ABB RobotStudio station: Oke_Iyanuoluwa.rspag

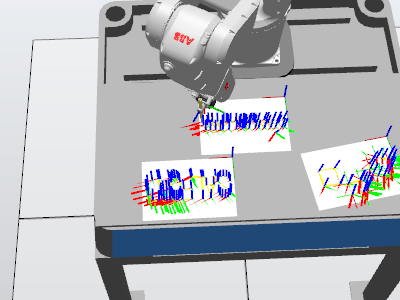
--- station ---
Station Project8 (saved by RobotStudio 24.1.10713.1)
Controller IRB1200_5_90, task T_ROB1: task frame (RAPID world) sits at (0, 233, 928) mm, rotated rx 0 ry 0 rz -90 deg in the station
Controller IRB1200_5_90
  mechanical unit ROB_1: IRB1200FPL_5_90_STD_02, 6 joints, base frame (0, 0, 0) mm
Layout (positions relative to the parent item):
  - IRB1200FPL_5_90_STD_02 [mechanism, from %ABB.RobotStudio.Models.IRB1200%\IRB1200FPL_5_90_STD_02.rslib] at (0, 233, 928) mm, rotated rx 0 ry 0 rz -90 deg; joint values [-0.5118, 1.2481, 0.7456, 0.0144, -1.9002, 0.0022] (rad or m)
  - Hardware [part], size 1120 x 955 x 931 mm
  - Pen for irb1200_2 [part] at (-177.12, -80.05, 1033) mm, rotated rx -87.72 ry 84.63 rz 62.19 deg, size 168 x 34 x 40 mm
  - IYANU2 [part] at (97, -87.87, 931) mm, rotated rx 0 ry 0 rz 180 deg, size 276.3 x 33.8 x 1 mm
Attachment: Pen for irb1200_2 is attached to IRB1200FPL_5_90_STD_02 / Link6
Targets, tools, work objects and paths stored in the station and not in the controller backup, written as RAPID:
! task T_ROB1
MODULE Module1
  PROC Shape_CircleCopy()
    MoveJ il_186,v100,fine,toolPen\WObj:=wobjShapes;
    MoveL il_187,v100,fine,toolPen\WObj:=wobjShapes;
    MoveL il_188,v100,fine,toolPen\WObj:=wobjShapes;
    MoveL il_189,v100,fine,toolPen\WObj:=wobjShapes;
    MoveL il_190,v100,fine,toolPen\WObj:=wobjShapes;
    MoveL il_191,v100,fine,toolPen\WObj:=wobjShapes;
    MoveL il_192,v100,fine,toolPen\WObj:=wobjShapes;
    MoveL il_193,v100,fine,toolPen\WObj:=wobjShapes;
    MoveL il_194,v100,fine,toolPen\WObj:=wobjShapes;
    MoveL il_195,v100,fine,toolPen\WObj:=wobjShapes;
    MoveL il_196,v100,fine,toolPen\WObj:=wobjShapes;
    MoveL il_197,v100,fine,toolPen\WObj:=wobjShapes;
    MoveL il_198,v100,fine,toolPen\WObj:=wobjShapes;
    MoveL il_199,v100,fine,toolPen\WObj:=wobjShapes;
  ENDPROC
ENDMODULE


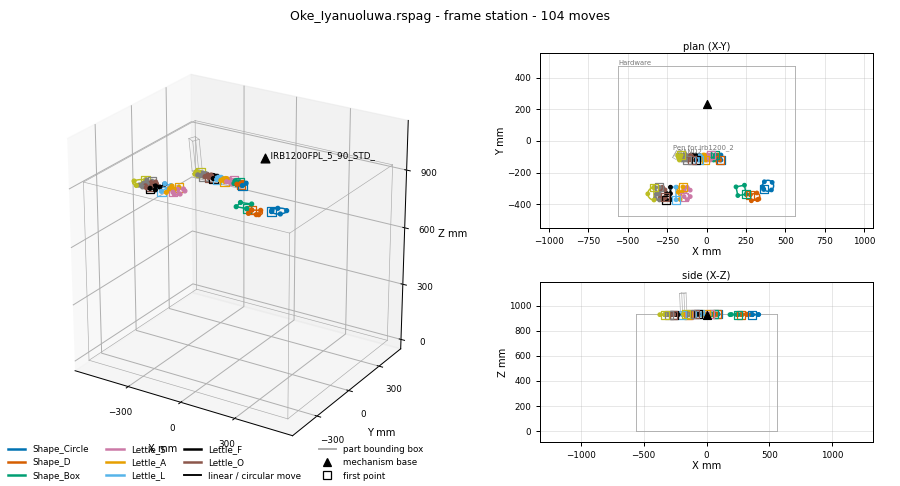
[picture p0: tool path of Oke_Iyanuoluwa.rspag in frame station, 104 of 104 moves have a stored position in this frame; points joined in program order, loops and branches not executed]
--- Controller Data/IRB1200_5_90/RAPID/TASK1/PROGMOD/Module1.mod ---
MODULE Module1
	TASK PERS tooldata toolPen:=[TRUE,[[100,0,20],[0.653281482,0.27059805,-0.653281482,-0.27059805]],[0.1,[50,0,10],[1,0,0,0],0,0,0]];
	TASK PERS wobjdata wobjShapes:=[FALSE,TRUE,"",[[403.87242208,428.126413661,0.1],[0.765935658,-0.001715767,0.001440186,-0.64291333]],[[0,0,0],[1,0,0,0]]];
	TASK PERS wobjdata wobjSalford:=[FALSE,TRUE,"",[[459.660289856,-90.375541036,0.1],[0.711712441,0,0,-0.702470925]],[[0,0,0],[1,0,0,0]]];
	TASK PERS wobjdata wobjName:=[FALSE,TRUE,"",[[234.420012927,103.808224608,3],[0.710975028,0,0,-0.703217256]],[[0,0,0],[1,0,0,0]]];
	VAR num MyChoice:=0;
    CONST robtarget Target_10:=[[511.467625969,422.116161374,0.1],[0,-0.087155742,0.996194698,0],[0,0,0,0],[9E+09,9E+09,9E+09,9E+09,9E+09,9E+09]];
    CONST robtarget Target_20:=[[485.422114903,400.261382644,0.1],[0,-0.573576436,0.819152044,0],[0,0,0,0],[9E+09,9E+09,9E+09,9E+09,9E+09,9E+09]];
    CONST robtarget Target_30:=[[491.326152944,366.777919042,0.1],[0,0.906307787,-0.422618262,0],[0,0,0,0],[9E+09,9E+09,9E+09,9E+09,9E+09,9E+09]];
    CONST robtarget Target_40:=[[523.275702051,355.149234169,0.1],[0,0.996194698,0.087155742,0],[0,0,0,0],[9E+09,9E+09,9E+09,9E+09,9E+09,9E+09]];
    CONST robtarget Target_50:=[[549.321213117,377.004012898,0.1],[0,0.819152044,0.573576436,0],[0,0,0,0],[9E+09,9E+09,9E+09,9E+09,9E+09,9E+09]];
    CONST robtarget Target_60:=[[543.417175076,410.4874765,0.1],[0,0.422618262,0.906307787,0],[0,0,0,0],[9E+09,9E+09,9E+09,9E+09,9E+09,9E+09]];
    CONST robtarget Target_70:=[[511.467625969,422.116161374,0.1],[0,-0.087155742,0.996194698,0],[0,0,0,0],[9E+09,9E+09,9E+09,9E+09,9E+09,9E+09]];
    CONST robtarget Target_80:=[[511.467625969,422.116161374,0.1],[0,-0.087155742,0.996194698,0],[0,0,0,0],[9E+09,9E+09,9E+09,9E+09,9E+09,9E+09]];
    CONST robtarget Target_90:=[[483.888200408,382.72865973,0.1],[0,0.766044443,-0.642787609,0],[0,0,0,0],[9E+09,9E+09,9E+09,9E+09,9E+09,9E+09]];
    CONST robtarget Target_100:=[[523.275702051,355.149234169,0.1],[0,0.996194698,0.087155742,0],[0,0,0,0],[9E+09,9E+09,9E+09,9E+09,9E+09,9E+09]];
    CONST robtarget Target_110:=[[550.855127612,394.536735812,0.1],[0,0.642787609,0.766044443,0],[0,0,0,0],[9E+09,9E+09,9E+09,9E+09,9E+09,9E+09]];
    CONST robtarget Target_120:=[[511.467625969,422.116161374,0.1],[0,-0.087155742,0.996194698,0],[0,0,0,0],[9E+09,9E+09,9E+09,9E+09,9E+09,9E+09]];
    CONST robtarget Target_130:=[[24.567771359,104.924042365,0.470081631],[0.001584245,-0.707222542,0.706987453,0.001583718],[0,0,0,0],[9E+09,9E+09,9E+09,9E+09,9E+09,9E+09]];
    CONST robtarget Target_140:=[[92.567767601,104.946649893,0.470182963],[0.001584245,-0.707222542,0.706987453,0.001583718],[0,0,0,0],[9E+09,9E+09,9E+09,9E+09,9E+09,9E+09]];
    CONST robtarget Target_150:=[[31.05454894,124.910653298,0.569625926],[0.001995763,-0.890928808,-0.454137469,-0.001017311],[0,0,0,0],[9E+09,9E+09,9E+09,9E+09,9E+09,9E+09]];
    CONST robtarget Target_160:=[[69.063596083,137.274389626,0.625018071],[0.002212567,-0.987711853,0.156269884,0.000350059],[0,0,0,0],[9E+09,9E+09,9E+09,9E+09,9E+09,9E+09]];
    CONST robtarget Target_170:=[[92.567767601,104.946605091,0.480182863],[0.001584245,-0.707222542,0.706987453,0.001583718],[0,0,0,0],[9E+09,9E+09,9E+09,9E+09,9E+09,9E+09]];
    CONST robtarget Target_180:=[[138.556128715,139.961590026,0.627057236],[0.002240087,-0.999997477,-0.000166233,-0.000000373],[0,0,0,0],[9E+09,9E+09,9E+09,9E+09,9E+09,9E+09]];
    CONST robtarget Target_190:=[[178.556126504,139.974888571,0.627116843],[0.002240087,-0.999997477,-0.000166233,-0.000000373],[0,0,0,0],[9E+09,9E+09,9E+09,9E+09,9E+09,9E+09]];
    CONST robtarget Target_200:=[[178.542827825,179.974484922,0.806323386],[0.001583718,-0.706987453,-0.707222542,-0.001584245],[0,0,0,0],[9E+09,9E+09,9E+09,9E+09,9E+09,9E+09]];
    CONST robtarget Target_210:=[[138.542830036,179.961186376,0.806263778],[0.000000373,-0.000166233,0.999997477,0.002240087],[0,0,0,0],[9E+09,9E+09,9E+09,9E+09,9E+09,9E+09]];
    CONST robtarget Target_220:=[[118.549480481,159.954738929,0.716630704],[0.001584245,-0.707222542,0.706987453,0.001583718],[0,0,0,0],[9E+09,9E+09,9E+09,9E+09,9E+09,9E+09]];
    CONST robtarget Target_230:=[[124.412046326,145.814693543,0.653280352],[0.002069714,-0.923940816,0.382528888,0.0008569],[0,0,0,0],[9E+09,9E+09,9E+09,9E+09,9E+09,9E+09]];
    CONST robtarget Target_240:=[[138.556128715,139.961590026,0.627057236],[0.002240087,-0.999997477,-0.000166233,-0.000000373],[0,0,0,0],[9E+09,9E+09,9E+09,9E+09,9E+09,9E+09]];
	CONST zonedata zone1:=[FALSE,50,75,75,7.5,75,7.5];
    !***********************************************************
    !
    ! Module:  Module1
    !
    ! Description:
    !   <Insert description here>
    !
    ! Author: sdp562
    !
    ! Version: 1.0
    !
    !***********************************************************


    !***********************************************************
    !
    ! Procedure main
    !
    !   This is the entry point of your program
    !
    !***********************************************************
    PROC main()
        TPErase;
        TPWrite "ABB RobotStudio Assignment - Oke Iyanuoluwa E.";
        TPReadFK MyChoice, "What will you like to draw/write?", "Shapes", "Salford", "MyName", "All of the above", stEmpty;
        TEST MyChoice
        CASE 1:
        	Shapes;
        CASE 2:
        	Salford;
        CASE 3:
        	MyName;
        CASE 4:
        	All;
        ENDTEST
    ENDPROC
	PROC Shapes()
		Shape_Circle;
		WaitTime 2;
		Shape_D;
		WaitTime 2;
		Shape_Box;
	ENDPROC
	PROC Salford()
		Lettle_S;
		Lettle_A;
		Lettle_L;
		Lettle_F;
		Lettle_O;
		Lettle_R;
		Lettle_D;
	ENDPROC
	PROC MyName()
		Letter_I;
		Letter_Y;
		Letter_A2;
		Letter_N;
		Letter_U;
		Letter_O2;
		Letter_L2;
		Letter_U2;
		Lettter_W;
		Letter_A3;
	ENDPROC
	PROC All()
		Shapes;
		WaitTime 2;
		Salford;
		WaitTime 2;
		MyName;
	ENDPROC
	PROC Shape_Circle()
		MoveJ [[88.31,121.43,0.9],[0.824392,-0.00205287,-0.000613241,0.566015],[0,-1,-1,1],[9E+09,9E+09,9E+09,9E+09,9E+09,9E+09]], v100, fine, toolPen\WObj:=wobjShapes;
		MoveC [[92.64,104.84,0.86],[0.823057,-0.0156436,0.0018724,0.567741],[0,-1,-1,1],[9E+09,9E+09,9E+09,9E+09,9E+09,9E+09]], [[75.99,75.44,-0.17],[0.809935,-0.0315414,0.00398667,0.585658],[0,-1,-1,1],[9E+09,9E+09,9E+09,9E+09,9E+09,9E+09]], v100, z10, toolPen\WObj:=wobjShapes;
		MoveC [[58.82,69.88,0.86],[0.801435,-0.0289154,0.00307954,0.597375],[0,-1,-1,1],[9E+09,9E+09,9E+09,9E+09,9E+09,9E+09]], [[27.99,88.04,1.08],[0.793128,-0.0040181,-0.000672612,0.609041],[0,-1,-1,1],[9E+09,9E+09,9E+09,9E+09,9E+09,9E+09]], v100, z10, toolPen\WObj:=wobjShapes;
		MoveC [[22.52,102.18,2.75],[0.794173,0.00861844,-0.00234434,0.607627],[0,-1,-1,1],[9E+09,9E+09,9E+09,9E+09,9E+09,9E+09]], [[41.05,134.37,1.12],[0.808041,0.0241329,-0.00490428,0.588611],[0,-1,-1,1],[9E+09,9E+09,9E+09,9E+09,9E+09,9E+09]], v100, z10, toolPen\WObj:=wobjShapes;
		MoveC [[57.78,139.03,0.62],[0.815418,0.0212852,-0.00468144,0.578462],[0,-1,-1,1],[9E+09,9E+09,9E+09,9E+09,9E+09,9E+09]], [[88.04,122.04,0.46],[0.826354,-0.00524432,0.00563442,0.563098],[0,0,0,1],[9E+09,9E+09,9E+09,9E+09,9E+09,9E+09]], v100, z10, toolPen\WObj:=wobjShapes;
		MoveL [[92.89,104.88,1.07],[0.825128,-0.0192408,0.00814959,0.564559],[0,0,0,1],[9E+09,9E+09,9E+09,9E+09,9E+09,9E+09]], v100, fine, toolPen\WObj:=wobjShapes;
	ENDPROC
	PROC Shape_D()
		MoveJ [[178.33,139.97,0.82],[0.862322,-0.0124094,0.00252986,0.506202],[0,-1,-1,1],[9E+09,9E+09,9E+09,9E+09,9E+09,9E+09]], v100, fine, toolPen\WObj:=wobjShapes;
		MoveL [[135.18,137.21,5.02],[0.84537,-0.00306398,-0.00014847,0.534173],[0,-1,-1,1],[9E+09,9E+09,9E+09,9E+09,9E+09,9E+09]], v100, fine, toolPen\WObj:=wobjShapes;
		MoveC [[122.15,149.76,0.21],[0.842062,0.00867023,-0.00276849,0.539304],[0,-1,-1,1],[9E+09,9E+09,9E+09,9E+09,9E+09,9E+09]],[[129.21,176.92,0.5],[0.84799,0.027547,-0.00720098,0.529246],[0,-1,-1,1],[9E+09,9E+09,9E+09,9E+09,9E+09,9E+09]],v100,z10,toolPen\WObj:=wobjShapes;
		MoveL [[139.7,179.86,0.26],[0.852174,0.027013,-0.00727031,0.52251],[0,-1,-1,1],[9E+09,9E+09,9E+09,9E+09,9E+09,9E+09]],v100,fine,toolPen\WObj:=wobjShapes;
		MoveL [[177.84,179.74,0.48],[0.866093,0.0181024,-0.00553464,0.499525],[0,-1,-1,1],[9E+09,9E+09,9E+09,9E+09,9E+09,9E+09]], v100, fine, toolPen\WObj:=wobjShapes;
		MoveL [[177.74,140.56,0.46],[0.862166,-0.0119302,0.00239961,0.50648],[0,-1,-1,1],[9E+09,9E+09,9E+09,9E+09,9E+09,9E+09]], v100, fine, toolPen\WObj:=wobjShapes;
	ENDPROC
	PROC Shape_Box()
		MoveJ [[203.77,133.76,1.09],[0.871331,-0.0217624,0.00553483,0.490182],[0,-1,-1,1],[9E+09,9E+09,9E+09,9E+09,9E+09,9E+09]], v100, fine, toolPen\WObj:=wobjShapes;
		MoveL [[256.61,132.45,1.81],[0.890805,-0.0302163,0.00946486,0.45328],[0,-1,-1,1],[9E+09,9E+09,9E+09,9E+09,9E+09,9E+09]], v100, fine, toolPen\WObj:=wobjShapes;
		MoveL [[258.42,76.19,0.13],[0.885765,-0.0735338,0.0230334,0.457692],[0,-1,-1,1],[9E+09,9E+09,9E+09,9E+09,9E+09,9E+09]], v100, fine, toolPen\WObj:=wobjShapes;
		MoveL [[203.82,75.03,0.64],[0.863466,-0.0662649,0.0170718,0.499743],[0,-1,-1,1],[9E+09,9E+09,9E+09,9E+09,9E+09,9E+09]], v100, fine, toolPen\WObj:=wobjShapes;
		MoveL [[203.76,134.33,0.29],[0.871385,-0.0215486,0.00547808,0.490096],[0,-1,-1,1],[9E+09,9E+09,9E+09,9E+09,9E+09,9E+09]], v100, fine, toolPen\WObj:=wobjShapes;
	ENDPROC
	PROC Lettle_S()
		MoveJ [[53.37,125.02,0.18],[0.963615,-0.0368758,0.0208919,0.263911],[-1,-1,-1,1],[9E+09,9E+09,9E+09,9E+09,9E+09,9E+09]], v100, fine, toolPen\WObj:=wobjSalford;
		MoveC [[49.77,135.43,-0.38],[0.962565,-0.0306315,0.0171276,0.268771],[-1,-1,-1,1],[9E+09,9E+09,9E+09,9E+09,9E+09,9E+09]],[[33.43,144.4,0.22],[0.958673,-0.0271208,0.0146305,0.282836],[-1,-1,-1,1],[9E+09,9E+09,9E+09,9E+09,9E+09,9E+09]],v100,z10,toolPen\WObj:=wobjSalford;
		MoveC [[24.37,142.14,-0.7],[0.956604,-0.0303515,0.0161234,0.289358],[-1,-1,-1,1],[9E+09,9E+09,9E+09,9E+09,9E+09,9E+09]],[[14.25,125.41,-0.8],[0.954383,-0.0435766,0.0229035,0.294497],[-1,-1,-1,1],[9E+09,9E+09,9E+09,9E+09,9E+09,9E+09]],v100,z10,toolPen\WObj:=wobjSalford;
		MoveL [[52.61,85.48,0.05],[0.963977,-0.0634662,0.0367473,0.255677],[-1,-1,-1,1],[9E+09,9E+09,9E+09,9E+09,9E+09,9E+09]], v100, fine, toolPen\WObj:=wobjSalford;
		MoveC [[50.58,75.89,-0.86],[0.963497,-0.070496,0.0408837,0.255014],[-1,-1,-1,1],[9E+09,9E+09,9E+09,9E+09,9E+09,9E+09]], [[33.64,65.84,-0.65],[0.959249,-0.0807602,0.0455016,0.266923],[-1,-1,-1,1],[9E+09,9E+09,9E+09,9E+09,9E+09,9E+09]], v100, z10, toolPen\WObj:=wobjSalford;
		MoveC [[24.01,68.64,-0.57],[0.956773,-0.0808116,0.0445486,0.275809],[-1,-1,-1,1],[9E+09,9E+09,9E+09,9E+09,9E+09,9E+09]], [[13.83,84.72,0.25],[0.954272,-0.0714944,0.0382654,0.28773],[-1,-1,-1,1],[9E+09,9E+09,9E+09,9E+09,9E+09,9E+09]], v100, z10, toolPen\WObj:=wobjSalford;
	ENDPROC
	PROC Lettle_A()
		MoveJ [[59.29,63.59,0.56],[0.965584,-0.0761666,0.0452825,0.244532],[-1,-1,-1,1],[9E+09,9E+09,9E+09,9E+09,9E+09,9E+09]], v100, fine, toolPen\WObj:=wobjSalford;
		MoveL [[78.48,142.56,0.21],[0.968312,-0.0201088,0.0117518,0.248656],[-1,-1,-1,1],[9E+09,9E+09,9E+09,9E+09,9E+09,9E+09]], v100, fine, toolPen\WObj:=wobjSalford;
		MoveL [[97.6,65.33,0.08],[0.973898,-0.0654568,0.0418275,0.213279],[-1,-1,-1,1],[9E+09,9E+09,9E+09,9E+09,9E+09,9E+09]], v100, fine, toolPen\WObj:=wobjSalford;
		MoveL [[89.96,96.6,-0.46],[0.971904,-0.0478143,0.0294838,0.228577],[-1,-1,-1,1],[9E+09,9E+09,9E+09,9E+09,9E+09,9E+09]], v100, fine, toolPen\WObj:=wobjSalford;
		MoveL [[66.19,95.41,0.1],[0.966964,-0.0539454,0.0318698,0.247092],[-1,-1,-1,1],[9E+09,9E+09,9E+09,9E+09,9E+09,9E+09]], v100, fine, toolPen\WObj:=wobjSalford;
	ENDPROC
	PROC Lettle_L()
		MoveJ [[104.07,144.38,0.11],[0.97299,-0.0134348,0.00814553,0.230311],[-1,-1,-1,1],[9E+09,9E+09,9E+09,9E+09,9E+09,9E+09]], v100, fine, toolPen\WObj:=wobjSalford;
		MoveL [[104.04,64.44,0.45],[0.975186,-0.0641498,0.0415036,0.207783],[-1,-1,-1,1],[9E+09,9E+09,9E+09,9E+09,9E+09,9E+09]], v100, fine, toolPen\WObj:=wobjSalford;
		MoveL [[137.15,65.07,3.55],[0.98121,-0.0534444,0.03662,0.181739],[-1,-1,-1,1],[9E+09,9E+09,9E+09,9E+09,9E+09,9E+09]], v100, fine, toolPen\WObj:=wobjSalford;
	ENDPROC
	PROC Lettle_F()
		MoveJ [[168.45,142.39,0.47],[0.982868,0.00146233,-0.00116288,0.184302],[-1,-1,-1,1],[9E+09,9E+09,9E+09,9E+09,9E+09,9E+09]], v100, fine, toolPen\WObj:=wobjSalford;
		MoveL [[138.89,143.45,-0.22],[0.978706,-0.00579302,0.00363048,0.205151],[-1,-1,-1,1],[9E+09,9E+09,9E+09,9E+09,9E+09,9E+09]], v100, fine, toolPen\WObj:=wobjSalford;
		MoveL [[138.71,64.53,0.13],[0.981408,-0.0541674,0.0372314,0.180327],[-1,-1,-1,1],[9E+09,9E+09,9E+09,9E+09,9E+09,9E+09]], v100, fine, toolPen\WObj:=wobjSalford;
		MoveL [[139.2,104.9,0.04],[0.980441,-0.0297577,0.0198081,0.19354],[-1,-1,-1,1],[9E+09,9E+09,9E+09,9E+09,9E+09,9E+09]], v100, fine, toolPen\WObj:=wobjSalford;
		MoveL [[163.35,104.29,0.13],[0.98403,-0.0232892,0.0160867,0.175739],[-1,-1,-1,1],[9E+09,9E+09,9E+09,9E+09,9E+09,9E+09]], v100, fine, toolPen\WObj:=wobjSalford;
	ENDPROC
	PROC Lettle_O()
		MoveJ [[173.96,128.87,0.16],[0.984312,-0.00540983,0.00360863,0.176314],[-1,-1,-1,1],[9E+09,9E+09,9E+09,9E+09,9E+09,9E+09]], v100, fine, toolPen\WObj:=wobjSalford;
		MoveL [[173.94,80.44,0.21],[0.986284,-0.0341024,0.0244644,0.15963],[-1,-1,-1,1],[9E+09,9E+09,9E+09,9E+09,9E+09,9E+09]], v100, fine, toolPen\WObj:=wobjSalford;
		MoveC [[175.45,72.54,0.15],[0.986703,-0.0381699,0.0276401,0.15555],[-1,-1,-1,1],[9E+09,9E+09,9E+09,9E+09,9E+09,9E+09]],[[188.93,64.2,0.43],[0.988644,-0.0384221,0.0286105,0.142433],[-1,-1,-1,1],[9E+09,9E+09,9E+09,9E+09,9E+09,9E+09]],v100,z10,toolPen\WObj:=wobjSalford;
		MoveC [[195.77,65.58,1.07],[0.989443,-0.0352391,0.0264717,0.138056],[-1,-1,-1,1],[9E+09,9E+09,9E+09,9E+09,9E+09,9E+09]], [[203.27,80.54,0.14],[0.989852,-0.0246889,0.018474,0.138713],[-1,-1,-1,1],[9E+09,9E+09,9E+09,9E+09,9E+09,9E+09]], v100, z10, toolPen\WObj:=wobjSalford;
		MoveL [[203.53,128.76,0.77],[0.987719,0.00330746,-0.00256956,0.156184],[-1,-1,-1,1],[9E+09,9E+09,9E+09,9E+09,9E+09,9E+09]], v100, fine, toolPen\WObj:=wobjSalford;
		MoveC [[201.3,136.66,-0.03],[0.987025,0.00719607,-0.00535274,0.160313],[-1,-1,-1,1],[9E+09,9E+09,9E+09,9E+09,9E+09,9E+09]],[[188.31,143.82,0.05],[0.985174,0.00778206,-0.00564351,0.171286],[-1,-1,-1,1],[9E+09,9E+09,9E+09,9E+09,9E+09,9E+09]],v100,z10,toolPen\WObj:=wobjSalford;
		MoveC [[181.27,142.39,0.1],[0.984448,0.00491604,-0.00359201,0.175572],[-1,-1,-1,1],[9E+09,9E+09,9E+09,9E+09,9E+09,9E+09]],[[173.94,129.74,-0.14],[0.984265,-0.00495753,0.00329245,0.176596],[-1,-1,-1,1],[9E+09,9E+09,9E+09,9E+09,9E+09,9E+09]],v100,z10,toolPen\WObj:=wobjSalford;
	ENDPROC
	PROC Lettle_R()
		MoveJ [[208.79,64.88,-0.01],[0.990914,-0.0315027,0.0241279,0.128514],[-1,-1,-1,1],[9E+09,9E+09,9E+09,9E+09,9E+09,9E+09]], v100, fine, toolPen\WObj:=wobjSalford;
		MoveL [[209.08,144.44,-0.05],[0.987319,0.0142011,-0.0104622,0.157764],[-1,-1,-1,1],[9E+09,9E+09,9E+09,9E+09,9E+09,9E+09]], v100, fine, toolPen\WObj:=wobjSalford;
		MoveC [[219.16,144.35,-0.36],[0.988273,0.0171204,-0.0127544,0.151196],[-1,-1,-1,1],[9E+09,9E+09,9E+09,9E+09,9E+09,9E+09]],[[235.25,134.7,-0.21],[0.990277,0.0164178,-0.0125916,0.137563],[-1,-1,-1,1],[9E+09,9E+09,9E+09,9E+09,9E+09,9E+09]],v100,z10,toolPen\WObj:=wobjSalford;
		MoveC [[237.91,124.53,-0.22],[0.991117,0.0113573,-0.0088594,0.132211],[-1,-1,-1,1],[9E+09,9E+09,9E+09,9E+09,9E+09,9E+09]], [[228.68,107.75,-0.12],[0.991253,-0.00118176,0.000738579,0.131966],[-1,-1,-1,1],[9E+09,9E+09,9E+09,9E+09,9E+09,9E+09]], v100, z10, toolPen\WObj:=wobjSalford;
		MoveL [[217.55,105.3,-0.37],[0.990341,-0.00622457,0.00453715,0.138436],[-1,-1,-1,1],[9E+09,9E+09,9E+09,9E+09,9E+09,9E+09]],v100,fine,toolPen\WObj:=wobjSalford;
		MoveL [[208.79,105.3,-0.1],[0.989466,-0.00895755,0.00651908,0.144342],[-1,-1,-1,1],[9E+09,9E+09,9E+09,9E+09,9E+09,9E+09]],v100,fine,toolPen\WObj:=wobjSalford;
		MoveL [[217.55,105.3,-0.37],[0.990341,-0.00622457,0.00453715,0.138436],[-1,-1,-1,1],[9E+09,9E+09,9E+09,9E+09,9E+09,9E+09]],v100,fine,toolPen\WObj:=wobjSalford;
		MoveL [[237.65,64.85,-0.41],[0.993699,-0.0216227,0.0172102,0.108617],[-1,-1,-1,1],[9E+09,9E+09,9E+09,9E+09,9E+09,9E+09]], v100, fine, toolPen\WObj:=wobjSalford;
	ENDPROC
	PROC Lettle_D()
		MoveJ [[243.84,64.96,0.21],[0.994217,-0.019248,0.0154319,0.104522],[-1,-1,-1,1],[9E+09,9E+09,9E+09,9E+09,9E+09,9E+09]], v100, fine, toolPen\WObj:=wobjSalford;
		MoveL [[243.91,144.14,-0.36],[0.990301,0.0246922,-0.0189375,0.13541],[-1,-1,-1,1],[9E+09,9E+09,9E+09,9E+09,9E+09,9E+09]], v100, fine, toolPen\WObj:=wobjSalford;
		MoveC [[263.39,138.39,-0.02],[0.991986,0.0277109,-0.0218618,0.121317],[-1,-1,-1,1],[9E+09,9E+09,9E+09,9E+09,9E+09,9E+09]],[[282.8,104.85,-0.3],[0.995125,0.0155247,-0.0129639,0.096522],[-1,-1,-1,1],[9E+09,9E+09,9E+09,9E+09,9E+09,9E+09]],v100,z10,toolPen\WObj:=wobjSalford;
		MoveC [[277.65,85.66,-0.51],[0.995778,0.00344946,-0.00304303,0.0916801],[-1,-1,-1,1],[9E+09,9E+09,9E+09,9E+09,9E+09,9E+09]],[[243.68,65.4,-0.35],[0.994187,-0.0191951,0.0153793,0.10482],[-1,-1,-1,1],[9E+09,9E+09,9E+09,9E+09,9E+09,9E+09]],v100,z10,toolPen\WObj:=wobjSalford;
	ENDPROC
	PROC Letter_I()
		MoveJ [[13.72,119.65,0.59],[0.868098,-0.0599828,0.00870245,0.492678],[0,-1,-1,1],[9E+09,9E+09,9E+09,9E+09,9E+09,9E+09]], v100, fine, toolPen\WObj:=wobjName;
		MoveL [[13.33,87.36,0.63],[0.859887,-0.0893615,0.0157035,0.502357],[0,-1,-1,1],[9E+09,9E+09,9E+09,9E+09,9E+09,9E+09]], v100, fine, toolPen\WObj:=wobjName;
	ENDPROC
	PROC Letter_Y()
		MoveJ [[21.84,119.55,0.46],[0.873255,-0.0617286,0.00988213,0.483237],[0,-1,-1,1],[9E+09,9E+09,9E+09,9E+09,9E+09,9E+09]], v100, fine, toolPen\WObj:=wobjName;
		MoveL [[32.44,102.18,0.7],[0.876528,-0.0793813,0.0157755,0.474499],[0,-1,-1,1],[9E+09,9E+09,9E+09,9E+09,9E+09,9E+09]],v100,fine,toolPen\WObj:=wobjName;
		MoveL [[43.89,119.16,0.67],[0.887013,-0.0655163,0.0130404,0.456886],[0,-1,-1,1],[9E+09,9E+09,9E+09,9E+09,9E+09,9E+09]], v100, fine, toolPen\WObj:=wobjName;
		MoveL [[32.44,102.18,0.7],[0.876528,-0.0793813,0.0157755,0.474499],[0,-1,-1,1],[9E+09,9E+09,9E+09,9E+09,9E+09,9E+09]],v100,fine,toolPen\WObj:=wobjName;
		MoveL [[32.4,87.33,0.76],[0.873159,-0.0931383,0.0194359,0.478059],[0,-1,-1,1],[9E+09,9E+09,9E+09,9E+09,9E+09,9E+09]],v100,fine,toolPen\WObj:=wobjName;
	ENDPROC
	PROC Letter_A2()
		MoveJ [[48.5,87.15,0.67],[0.884104,-0.0956481,0.0226303,0.456836],[0,-1,-1,1],[9E+09,9E+09,9E+09,9E+09,9E+09,9E+09]],v100,fine,toolPen\WObj:=wobjName;
		MoveL [[60.07,119,0.6],[0.896847,-0.0673998,0.0152597,0.436909],[0,-1,-1,1],[9E+09,9E+09,9E+09,9E+09,9E+09,9E+09]],v100,fine,toolPen\WObj:=wobjName;
		MoveL [[67.08,99.31,0.54],[0.898341,-0.086007,0.022352,0.430216],[0,-1,-1,1],[9E+09,9E+09,9E+09,9E+09,9E+09,9E+09]], v100, fine, toolPen\WObj:=wobjName;
		MoveL [[52.8,99.2,0.56],[0.88923,-0.0849219,0.0200305,0.449062],[0,-1,-1,1],[9E+09,9E+09,9E+09,9E+09,9E+09,9E+09]],v100,fine,toolPen\WObj:=wobjName;
		MoveL [[67.08,99.31,0.54],[0.898341,-0.086007,0.022352,0.430216],[0,-1,-1,1],[9E+09,9E+09,9E+09,9E+09,9E+09,9E+09]], v100, fine, toolPen\WObj:=wobjName;
		MoveL [[71.13,86.94,0.76],[0.899026,-0.0976712,0.0269373,0.426013],[0,-1,-1,1],[9E+09,9E+09,9E+09,9E+09,9E+09,9E+09]], v100, fine, toolPen\WObj:=wobjName;
	ENDPROC
	PROC Letter_N()
		MoveJ [[78.86,86.85,0.53],[0.903952,-0.0980786,0.0283703,0.415267],[0,-1,-1,1],[9E+09,9E+09,9E+09,9E+09,9E+09,9E+09]], v100, fine, toolPen\WObj:=wobjName;
		MoveL [[80.35,118.78,0.63],[0.908747,-0.0687307,0.0178438,0.411261],[0,-1,-1,1],[9E+09,9E+09,9E+09,9E+09,9E+09,9E+09]], v100, fine, toolPen\WObj:=wobjName;
		MoveL [[99.92,86.42,0.81],[0.916899,-0.0981308,0.0319746,0.385544],[0,-1,-1,1],[9E+09,9E+09,9E+09,9E+09,9E+09,9E+09]], v100, fine, toolPen\WObj:=wobjName;
		MoveL [[100.41,118.30,0.70],[0.919934,-0.0691563,0.0201723,0.385399],[0,-1,-1,1],[9E+09,9E+09,9E+09,9E+09,9E+09,9E+09]], v100, fine, toolPen\WObj:=wobjName;
	ENDPROC
	PROC Letter_U()
		MoveJ [[111.23,118.87,0.50],[0.925756,-0.0682694,0.0209811,0.371316],[-1,-1,-1,1],[9E+09,9E+09,9E+09,9E+09,9E+09,9E+09]], v100, fine, toolPen\WObj:=wobjName;
		MoveL [[111.23,95.90,0.61],[0.924283,-0.0888486,0.0299018,0.370018],[-1,-1,-1,1],[9E+09,9E+09,9E+09,9E+09,9E+09,9E+09]], v100, fine, toolPen\WObj:=wobjName;
		MoveC [[112.75,90.34,0.72],[0.924719,-0.0937515,0.0322865,0.367509],[-1,-1,-1,1],[9E+09,9E+09,9E+09,9E+09,9E+09,9E+09]], [[117.49,86.79,0.66],[0.928903,-0.0893218,0.0336693,0.357808],[-1,0,-1,1],[9E+09,9E+09,9E+09,9E+09,9E+09,9E+09]], v100, z10, toolPen\WObj:=wobjName;
		MoveL [[124.93,86.60,0.61],[0.932986,-0.0886965,0.0345911,0.347092],[-1,0,-1,1],[9E+09,9E+09,9E+09,9E+09,9E+09,9E+09]], v100, fine, toolPen\WObj:=wobjName;
		MoveC [[127.95,88.29,0.51],[0.934698,-0.086822,0.0341999,0.342976],[-1,0,-1,1],[9E+09,9E+09,9E+09,9E+09,9E+09,9E+09]], [[131.79,95.94,0.50],[0.93703,-0.0794817,0.0312953,0.338643],[-1,0,-1,1],[9E+09,9E+09,9E+09,9E+09,9E+09,9E+09]], v100, z10, toolPen\WObj:=wobjName;
		MoveL [[132.14,117.92,0.42],[0.937827,-0.0600286,0.0221247,0.341156],[-1,0,-1,1],[9E+09,9E+09,9E+09,9E+09,9E+09,9E+09]], v100, fine, toolPen\WObj:=wobjName;
	ENDPROC
	PROC Letter_O2()
		MoveJ [[153.90,117.97,0.57],[0.947908,-0.0570213,0.0227871,0.31257],[-1,0,-1,1],[9E+09,9E+09,9E+09,9E+09,9E+09,9E+09]], v100, fine, toolPen\WObj:=wobjName;
		MoveC [[161.21,113.59,0.57],[0.951126,-0.0595025,0.0248193,0.301998],[-1,0,-1,1],[9E+09,9E+09,9E+09,9E+09,9E+09,9E+09]], [[164.13,107.24,0.57],[0.952446,-0.0643384,0.0277382,0.296543],[-1,0,-1,1],[9E+09,9E+09,9E+09,9E+09,9E+09,9E+09]], v100, z10, toolPen\WObj:=wobjName;
		MoveC [[164.61,101.96,0.57],[0.952696,-0.0687172,0.0301841,0.294511],[-1,0,-1,1],[9E+09,9E+09,9E+09,9E+09,9E+09,9E+09]], [[162.12,91.51,0.63],[0.951616,-0.0781205,0.0350085,0.295125],[-1,0,-1,1],[9E+09,9E+09,9E+09,9E+09,9E+09,9E+09]], v100, z10, toolPen\WObj:=wobjName;
		MoveC [[158.90,87.99,0.53],[0.950124,-0.0818456,0.0365588,0.298711],[-1,0,-1,1],[9E+09,9E+09,9E+09,9E+09,9E+09,9E+09]], [[149.58,86.32,0.53],[0.945671,-0.0851543,0.0368403,0.311604],[-1,0,-1,1],[9E+09,9E+09,9E+09,9E+09,9E+09,9E+09]], v100, z10, toolPen\WObj:=wobjName;
		MoveC [[145.30,89.01,0.48],[0.943632,-0.0835877,0.0353454,0.318313],[-1,0,-1,1],[9E+09,9E+09,9E+09,9E+09,9E+09,9E+09]], [[142.01,93.28,0.47],[0.943669,-0.0771096,0.0354276,0.319825],[-1,0,0,1],[9E+09,9E+09,9E+09,9E+09,9E+09,9E+09]], v100, z10, toolPen\WObj:=wobjName;
		MoveC [[140.96,103.97,0.57],[0.943374,-0.0678218,0.0307172,0.323268],[-1,0,0,1],[9E+09,9E+09,9E+09,9E+09,9E+09,9E+09]], [[144.24,114.09,0.50],[0.945023,-0.058511,0.026528,0.32063],[-1,0,0,1],[9E+09,9E+09,9E+09,9E+09,9E+09,9E+09]], v100, z10, toolPen\WObj:=wobjName;
		MoveC [[147.02,116.42,0.50],[0.946296,-0.0560756,0.0256059,0.317371],[-1,0,0,1],[9E+09,9E+09,9E+09,9E+09,9E+09,9E+09]], [[154.64,117.76,0.62],[0.949667,-0.0536972,0.0251428,0.307599],[-1,0,0,1],[9E+09,9E+09,9E+09,9E+09,9E+09,9E+09]], v100, z10, toolPen\WObj:=wobjName;
	ENDPROC
	PROC Letter_L2()
		MoveJ [[174.14,117.95,0.53],[0.957737,-0.0499267,0.0249432,0.28218],[-1,0,0,1],[9E+09,9E+09,9E+09,9E+09,9E+09,9E+09]], v100, fine, toolPen\WObj:=wobjName;
		MoveL [[173.69,86.16,0.75],[0.958093,-0.0765809,0.0398676,0.273136],[-1,0,0,1],[9E+09,9E+09,9E+09,9E+09,9E+09,9E+09]], v100, fine, toolPen\WObj:=wobjName;
		MoveL [[191.57,86.08,0.64],[0.965262,-0.0718343,0.0397509,0.248049],[-1,0,0,1],[9E+09,9E+09,9E+09,9E+09,9E+09,9E+09]], v100, fine, toolPen\WObj:=wobjName;
	ENDPROC
	PROC Letter_U2()
		MoveJ [[199.14,117.79,0.46],[0.966932,-0.0442837,0.0238707,0.250022],[-1,0,0,1],[9E+09,9E+09,9E+09,9E+09,9E+09,9E+09]], v100, fine, toolPen\WObj:=wobjName;
		MoveL [[199.22,92.97,0.61],[0.967892,-0.0640605,0.0359795,0.240391],[-1,0,0,1],[9E+09,9E+09,9E+09,9E+09,9E+09,9E+09]], v100, fine, toolPen\WObj:=wobjName;
		MoveC [[201.20,88.60,0.63],[0.968732,-0.0669487,0.0380785,0.235854],[-1,0,0,1],[9E+09,9E+09,9E+09,9E+09,9E+09,9E+09]], [[205.25,85.77,0.77],[0.970239,-0.067893,0.0392683,0.229097],[-1,0,0,1],[9E+09,9E+09,9E+09,9E+09,9E+09,9E+09]], v100, z10, toolPen\WObj:=wobjName;
		MoveC [[214.25,86.32,0.71],[0.97324,-0.0645685,0.0383544,0.21717],[-1,0,0,1],[9E+09,9E+09,9E+09,9E+09,9E+09,9E+09]], [[219.34,94.09,0.55],[0.974551,-0.0569651,0.0339195,0.214138],[-1,0,0,1],[9E+09,9E+09,9E+09,9E+09,9E+09,9E+09]], v100, z10, toolPen\WObj:=wobjName;
		MoveL [[219.86,117.45,0.58],[0.973582,-0.0388773,0.0221727,0.223909],[-1,0,0,1],[9E+09,9E+09,9E+09,9E+09,9E+09,9E+09]], v100, fine, toolPen\WObj:=wobjName;
	ENDPROC
	PROC Lettter_W()
		MoveJ [[227.45,117.32,0.57],[0.975801,-0.0367211,0.0213435,0.214496],[-1,0,0,1],[9E+09,9E+09,9E+09,9E+09,9E+09,9E+09]], v100, fine, toolPen\WObj:=wobjName;
		MoveL [[235.03,85.16,0.74],[0.97954,-0.0582023,0.0367607,0.189108],[-1,0,0,1],[9E+09,9E+09,9E+09,9E+09,9E+09,9E+09]], v100, fine, toolPen\WObj:=wobjName;
		MoveL [[244.00,117.10,0.60],[0.980228,-0.0317078,0.0191296,0.194374],[-1,0,0,1],[9E+09,9E+09,9E+09,9E+09,9E+09,9E+09]], v100, fine, toolPen\WObj:=wobjName;
		MoveL [[252.62,85.27,0.72],[0.984067,-0.0515249,0.0340638,0.166725],[-1,0,0,1],[9E+09,9E+09,9E+09,9E+09,9E+09,9E+09]], v100, fine, toolPen\WObj:=wobjName;
		MoveL [[260.92,116.76,0.54],[0.984206,-0.0263207,0.0163866,0.174289],[-1,0,0,1],[9E+09,9E+09,9E+09,9E+09,9E+09,9E+09]], v100, fine, toolPen\WObj:=wobjName;
	ENDPROC
	PROC Letter_A3()
		MoveJ [[265.08,84.93,0.61],[0.986887,-0.0469029,0.0319696,0.151105],[-1,0,0,1],[9E+09,9E+09,9E+09,9E+09,9E+09,9E+09]], v100, fine, toolPen\WObj:=wobjName;
		MoveL [[276.67,116.62,0.69],[0.987413,-0.0208441,0.0132138,0.156226],[-1,0,0,1],[9E+09,9E+09,9E+09,9E+09,9E+09,9E+09]], v100, fine, toolPen\WObj:=wobjName;
		MoveL [[283.50,96.71,0.74],[0.989868,-0.0316418,0.021767,0.136696],[-1,0,0,1],[9E+09,9E+09,9E+09,9E+09,9E+09,9E+09]], v100, fine, toolPen\WObj:=wobjName;
		MoveL [[269.74,96.85,0.63],[0.987257,-0.0369296,0.0247602,0.152796],[-1,0,0,1],[9E+09,9E+09,9E+09,9E+09,9E+09,9E+09]], v100, fine, toolPen\WObj:=wobjName;
		MoveL [[283.50,96.71,0.74],[0.989868,-0.0316418,0.021767,0.136696],[-1,0,0,1],[9E+09,9E+09,9E+09,9E+09,9E+09,9E+09]], v100, fine, toolPen\WObj:=wobjName;
		MoveL [[287.50,84.44,0.57],[0.991163,-0.0380666,0.0272334,0.124119],[-1,0,0,1],[9E+09,9E+09,9E+09,9E+09,9E+09,9E+09]], v100, fine, toolPen\WObj:=wobjName;
	ENDPROC
ENDMODULE

--- Controller Data/IRB1200_5_90/RAPID/TASK1/SYSMOD/LINKEDM.sys ---
%%%
  VERSION:1
  LANGUAGE:ENGLISH
%%%

MODULE LINKEDM (SYSMODULE)

! FOLLOWER
!     Name of electronically linked follower axis used by operator at teach pendent.
      PERS string l_f_axis_name{5}       :=  ["",  "", "", "", ""];

!     Name of the mechanical unit for follower axis.
      PERS string l_f_mecunt_n{5}  :=  ["", "", "", "", ""];

!     Linked follower axis number in the mechanical unit (first axis in mech. unit is number 1).
      PERS num l_f_axis_no{5}      :=  [0,          0,   0,  0,  0];

! MASTER
!     Name of the mechanical unit for linked master axis.
      PERS string l_m_mecunt_n{5} :=  ["", "", "", "", ""];

!     Linked master axis number in the mechanical unit (first axis in mech. unit is number 1).
!     See axis number table in documentation for different master mechanical units.
      PERS num l_m_axis_no{5}     :=  [0,  0,  0,  0,  0];

! POSITION OFFSET
!     The increase of the allowed offset position between the master and follower
!     positions, used when starting AUTO mode. As soon as the offset is decreased
!     the old configurated parameter is used.
!     Example: 3 => the configurated value of allowed offset is increased 3 times.
      PERS num offset_ratio{5}       :=  [10,  10,   10,  10,  10];

! SPEED RATIO
!     Speed_ratio used in AUTO and JOG modes [ very_slow   slow    normal    fast]
!     Value 1 = max allowed manual speed.
      CONST num speed_ratio {20}      := [0.01, 0.01, 0.01, 0.01, 0.01,
                                          0.05, 0.05, 0.05, 0.05, 0.05,
                                          0.20, 0.20, 0.20, 0.20, 0.20,
                                          1.00, 1.00, 1.00, 1.00, 1.00];

! STEP SIZE
!     Displacement position used in JOG mode for each activation of positive or
!     negative movement.                  [very_short    short   normal   long]
!     Unit degees or meter.
      CONST num displacement {20}     := [0.001, 0.001, 0.001, 0.001, 0.001,
                                          0.005, 0.005, 0.005, 0.005, 0.005,
                                          0.020, 0.020, 0.020, 0.020, 0.020,
                                          0.100, 0.100, 0.100, 0.100, 0.100];


!-------------------------------------------------------------
 PROC Linked_m ()
      Linked_m_exe ;
 ENDPROC
ENDMODULE
